// TIA Portal V20 export
VAR_GLOBAL   // PLC tag table "Unit1Em7"
   "BA030AZSBK22.00" AT %I1084.0 : Bool;   // SEPA GRIPPER CLAMP OPEN
   "BA030AZSBK22.03" AT %I1084.3 : Bool;   // SEPA GRIPPER BACKWARD
   "BA030AZSBK22.02" AT %I1084.2 : Bool;   // SEPA GRIPPER CLAMP DETECT SENSOR
   "BA030AZSBK22.10" AT %I1085.0 : Bool;   // SEPA GRIPPER CLAMP CLOSE
   "BA030AZSBK22.13" AT %I1085.3 : Bool;   // SEPA GRIPPER FORWARD
   "BA030AZSBK23.02" AT %I1088.2 : Bool;   // SEPA CUTTER UP
   "BA030AZSBK23.06" AT %I1088.6 : Bool;   // SEPA DETECT SENSOR
   "BA030AZSBK23.12" AT %I1089.2 : Bool;   // SEPA CUTTER DOWN
   "BA030AZSBK24.00" AT %I1092.0 : Bool;   // SEPA CLAMP TOP REAR UP
   "BA030AZSBK24.02" AT %I1092.2 : Bool;   // SEPA CLAMP TOP FRONT UP
   "BA030AZSBK24.04" AT %I1092.4 : Bool;   // SEPA CLAMP BTM REAR UP
   "BA030AZSBK24.06" AT %I1092.6 : Bool;   // SEPA CLAMP BTM FRONT UP
   "BA030AZSBK24.10" AT %I1093.0 : Bool;   // SEPA CLAMP TOP REAR DOWN
   "BA030AZSBK24.12" AT %I1093.2 : Bool;   // SEPA CLAMP TOP FRONT DOWN
   "BA030AZSBK24.14" AT %I1093.4 : Bool;   // SEPA CLAMP BTM REAR DOWN
   "BA030AZSBK24.16" AT %I1093.6 : Bool;   // SEPA CLAMP BTM FRONT DOWN
   "BA030AZSBK26.01" AT %I1100.1 : Bool;   // JR WINDER CLAMP TOP REAR UP/DOWN
   "BA030AZSBK26.03" AT %I1100.3 : Bool;   // JR WINDER CLAMP TOP FRONT UP/DOWN
   "BA030AZSBK26.05" AT %I1100.5 : Bool;   // JR WINDER CLAMP TOP REAR PRESSURE SWITCH
   "BA030AZSBK26.11" AT %I1101.1 : Bool;   // SPARE
   "BA030AZSBK26.13" AT %I1101.3 : Bool;   // SPARE
   "BA030AZSBK26.15" AT %I1101.5 : Bool;   // JR WINDER CLAMP TOP FRONT PRESSURE SWITCH
   "BA030AZSBK27.01" AT %I1104.1 : Bool;   // JR WINDER CLAMP BTM REAR UP/DOWN
   "BA030AZSBK27.03" AT %I1104.3 : Bool;   // JR WINDER CLAMP BTM FRONT UP/DOWN
   "BA030AZSBK27.05" AT %I1104.5 : Bool;   // JR WINDER CLAMP BTM REAR PRESSURE SWITCH
   "BA030AZSBK27.06" AT %I1104.6 : Bool;   // JR WINDER STACK DETECT SENSOR
   "BA030AZSBK27.11" AT %I1105.1 : Bool;   // SPARE
   "BA030AZSBK27.13" AT %I1105.3 : Bool;   // SPARE
   "BA030AZSBK27.15" AT %I1105.5 : Bool;   // JR WINDER CLAMP BTM FRONT PRESSURE SWITCH
   "BA030AZSBK28.02" AT %I1108.2 : Bool;   // PUSH ROLLER BACKWARD
   "BA030AZSBK28.03" AT %I1108.3 : Bool;   // PUSH ROLLER FORWARD
   "BA030AZSBK10.01" AT %I1036.1 : Bool;   // SEPA CLAMP SAFETY PIN DETECT SENSOR
   "BA030AZSBK10.11" AT %I1037.1 : Bool;   // SEPA GRIPPER SAFETY PIN DETECT SENSOR
   "BA030AZSBK10.03" AT %I1036.3 : Bool;   // SEPA CLAMP PRESSURE SWITCH
   "BA030AZSPM07.02" AT %Q2024.2 : Bool;   // JR WINDER CLAMP BTM REAR UP
   "BA030AZSPM07.03" AT %Q2024.3 : Bool;   // JR WINDER CLAMP BTM REAR DOWN
   "BA030AZSPM07.04" AT %Q2024.4 : Bool;   // JR WINDER CLAMP TOP FRONT UP
   "BA030AZSPM07.05" AT %Q2024.5 : Bool;   // JR WINDER CLAMP TOP FRONT DOWN
   "BA030AZSPM07.06" AT %Q2024.6 : Bool;   // JR WINDER CLAMP BTM FRONT UP
   "BA030AZSPM07.07" AT %Q2024.7 : Bool;   // JR WINDER CLAMP BTM FRONT DOWN
   "BA030AZSPM07.12" AT %Q2025.2 : Bool;   // PUSH ROLLER FORWARD
   "BA030AZSPM07.13" AT %Q2025.3 : Bool;   // PUSH ROLLER BACKWARD
   "BA030AZSPM03.00" AT %Q2008.0 : Bool;   // SEPA CUTTER FRONT&REAR DOWN
   "BA030AZSPM03.01" AT %Q2008.1 : Bool;   // SEPA CUTTER FRONT&REAR UP
   "BA030AZSPM03.02" AT %Q2008.2 : Bool;   // SEPA CLAMP TOP REAR DOWN
   "BA030AZSPM03.03" AT %Q2008.3 : Bool;   // SEPA CLAMP TOP REAR UP
   "BA030AZSPM03.04" AT %Q2008.4 : Bool;   // SEPA CLAMP TOP FRONT DOWN
   "BA030AZSPM03.05" AT %Q2008.5 : Bool;   // SEPA CLAMP TOP FRONT UP
   "BA030AZSPM03.06" AT %Q2008.6 : Bool;   // SEPA CLAMP BTM REAR DOWN
   "BA030AZSPM03.07" AT %Q2008.7 : Bool;   // SEPA CLAMP BTM REAR UP
   "BA030AZSPM03.10" AT %Q2009.0 : Bool;   // SEPA CLAMP BTM FRONT DOWN
   "BA030AZSPM03.11" AT %Q2009.1 : Bool;   // SEPA CLAMP BTM FRONT UP
   "BA030AZSPM03.12" AT %Q2009.2 : Bool;   // SEPA GRIPPER CLOSE
   "BA030AZSPM03.13" AT %Q2009.3 : Bool;   // SEPA GRIPPER OPEN
   "BA030AZSPM03.14" AT %Q2009.4 : Bool;   // SEPA GRIPPER FORWARD
   "BA030AZSPM03.15" AT %Q2009.5 : Bool;   // SEPA GRIPPER BACKWARD
   "BA030AZSPM07.00" AT %Q2024.0 : Bool;   // JR WINDER CLAMP TOP REAR UP
   "BA030AZSPM07.01" AT %Q2024.1 : Bool;   // JR WINDER CLAMP TOP REAR DOWN
END_VAR
VAR_GLOBAL CONSTANT   // user constants
   U1EM7_JOB01 : DInt := 1;
   U1EM7_JOB02 : DInt := 2;
   U1EM7_JOB03 : DInt := 3;
   U1EM7_JOB04 : DInt := 4;
   U1EM7_JOB05 : DInt := 5;
   U1EM7_JOB06 : DInt := 6;
   U1EM7_JOB07 : DInt := 7;
   U1EM7_JOB08 : DInt := 8;
   U1EM7_JOB09 : DInt := 9;
   U1EM7_JOB10 : DInt := 10;
   U1EM7_JOB11 : DInt := 11;
   U1EM7_JOB12 : DInt := 12;
   U1EM7_JOB13 : DInt := 13;
   U1EM7_JOB14 : DInt := 14;
   U1EM7_JOB15 : DInt := 15;
   U1EM7_JOB16 : DInt := 16;
   U1EM7_JOB17 : DInt := 17;
   U1EM7_JOB18 : DInt := 18;
   U1EM7_JOB19 : DInt := 19;
   U1EM7_JOB20 : DInt := 20;
   U1EM7_JOB21 : DInt := 21;
   U1EM7_JOB22 : DInt := 22;
   U1EM7_JOB23 : DInt := 23;
   U1EM7_JOB24 : DInt := 24;
   U1EM7_JOB25 : DInt := 25;
   U1EM7_JOB26 : DInt := 26;
   U1EM7_JOB27 : DInt := 27;
   U1EM7_JOB28 : DInt := 28;
   U1EM7_JOB29 : DInt := 29;
   U1EM7_JOB30 : DInt := 30;
   U1EM7_JOB31 : DInt := 31;
   U1EM7_JOB32 : DInt := 32;
   U1EM7_JOB33 : DInt := 33;
   U1EM7_JOB34 : DInt := 34;
   U1EM7_JOB35 : DInt := 35;
   U1EM7_JOB36 : DInt := 36;
   U1EM7_JOB37 : DInt := 37;
   U1EM7_JOB38 : DInt := 38;
   U1EM7_JOB39 : DInt := 39;
   U1EM7_JOB40 : DInt := 40;
   U1EM7_JOB41 : DInt := 41;
   U1EM7_JOB42 : DInt := 42;
   U1EM7_JOB43 : DInt := 43;
   U1EM7_JOB44 : DInt := 44;
   U1EM7_JOB45 : DInt := 45;
   U1EM7_JOB46 : DInt := 46;
   U1EM7_JOB47 : DInt := 47;
   U1EM7_JOB48 : DInt := 48;
   U1EM7_JOB49 : DInt := 49;
   U1EM7_JOB50 : DInt := 50;
   U1EM7_JOB51 : DInt := 51;
   U1EM7_JOB52 : DInt := 52;
   U1EM7_JOB53 : DInt := 53;
   U1EM7_JOB54 : DInt := 54;
   U1EM7_JOB55 : DInt := 55;
   U1EM7_JOB56 : DInt := 56;
   U1EM7_JOB57 : DInt := 57;
   U1EM7_JOB58 : DInt := 58;
   U1EM7_JOB59 : DInt := 59;
   U1EM7_JOB60 : DInt := 60;
   U1EM7_JOB61 : DInt := 61;
   U1EM7_JOB62 : DInt := 62;
   U1EM7_JOB63 : DInt := 63;
   U1EM7_JOB64 : DInt := 64;
   U1EM7_JOB65 : DInt := 65;
   U1EM7_JOB66 : DInt := 66;
   U1EM7_JOB67 : DInt := 67;
   U1EM7_JOB68 : DInt := 68;
   U1EM7_JOB69 : DInt := 69;
   U1EM7_JOB70 : DInt := 70;
   U1EM7_JOB71 : DInt := 71;
   U1EM7_JOB72 : DInt := 72;
   U1EM7_JOB73 : DInt := 73;
   U1EM7_JOB74 : DInt := 74;
   U1EM7_JOB75 : DInt := 75;
   U1EM7_JOB76 : DInt := 76;
   U1EM7_JOB77 : DInt := 77;
   U1EM7_JOB78 : DInt := 78;
   U1EM7_JOB79 : DInt := 79;
   U1EM7_JOB80 : DInt := 80;
   U1EM7_JOB81 : DInt := 81;
   U1EM7_JOB82 : DInt := 82;
   U1EM7_JOB83 : DInt := 83;
   U1EM7_JOB84 : DInt := 84;
   U1EM7_JOB85 : DInt := 85;
   U1EM7_JOB86 : DInt := 86;
   U1EM7_JOB87 : DInt := 87;
   U1EM7_JOB88 : DInt := 88;
   U1EM7_JOB89 : DInt := 89;
   U1EM7_JOB90 : DInt := 90;
   U1EM7_JOB91 : DInt := 91;
   U1EM7_JOB92 : DInt := 92;
   U1EM7_JOB93 : DInt := 93;
   U1EM7_JOB94 : DInt := 94;
   U1EM7_JOB95 : DInt := 95;
   U1EM7_JOB96 : DInt := 96;
   U1EM7_JOB97 : DInt := 97;
   U1EM7_JOB98 : DInt := 98;
   U1EM7_JOB99 : DInt := 99;
   U1EM7_SEQUENCE01 : Int := 1;
   U1EM7_SEQUENCE02 : Int := 2;
   U1EM7_SEQUENCE03 : Int := 3;
   U1EM7_SEQUENCE04 : Int := 4;
   U1EM7_SEQUENCE05 : Int := 5;
   U1EM7_SEQUENCE06 : Int := 6;
   U1EM7_SEQUENCE07 : Int := 7;
   U1EM7_SEQUENCE08 : Int := 8;
   U1EM7_SEQUENCE09 : Int := 9;
   U1EM7_SEQUENCE10 : Int := 10;
   U1EM7_SEQUENCE11 : Int := 11;
   U1EM7_SEQUENCE12 : Int := 12;
   U1EM7_SEQUENCE13 : Int := 13;
   U1EM7_SEQUENCE14 : Int := 14;
   U1EM7_SEQUENCE15 : Int := 15;
   U1EM7_SEQUENCE16 : Int := 16;
   U1EM7_SEQUENCE17 : Int := 17;
   U1EM7_SEQUENCE18 : Int := 18;
   U1EM7_SEQUENCE19 : Int := 19;
   U1EM7_SEQUENCE20 : Int := 20;
   U1EM7_SEQUENCE21 : Int := 21;
   U1EM7_SEQUENCE22 : Int := 22;
   U1EM7_SEQUENCE23 : Int := 23;
   U1EM7_SEQUENCE24 : Int := 24;
   U1EM7_SEQUENCE25 : Int := 25;
   U1EM7_SEQUENCE26 : Int := 26;
   U1EM7_SEQUENCE27 : Int := 27;
   U1EM7_SEQUENCE28 : Int := 28;
   U1EM7_SEQUENCE29 : Int := 29;
   U1EM7_SEQUENCE30 : Int := 30;
   U1EM7_SEQUENCE31 : Int := 31;
   U1EM7_SEQUENCE32 : Int := 32;
   U1EM7_SEQUENCE33 : Int := 33;
   U1EM7_SEQUENCE34 : Int := 34;
   U1EM7_SEQUENCE35 : Int := 35;
   U1EM7_SEQUENCE36 : Int := 36;
   U1EM7_SEQUENCE37 : Int := 37;
   U1EM7_SEQUENCE38 : Int := 38;
   U1EM7_SEQUENCE39 : Int := 39;
   U1EM7_SEQUENCE40 : Int := 40;
   U1EM7_SEQUENCE41 : Int := 41;
   U1EM7_SEQUENCE42 : Int := 42;
   U1EM7_SEQUENCE43 : Int := 43;
   U1EM7_SEQUENCE44 : Int := 44;
   U1EM7_SEQUENCE45 : Int := 45;
   U1EM7_SEQUENCE46 : Int := 46;
   U1EM7_SEQUENCE47 : Int := 47;
   U1EM7_SEQUENCE48 : Int := 48;
   U1EM7_SEQUENCE49 : Int := 49;
   U1EM7_SEQUENCE50 : Int := 50;
   U1EM7_SEQUENCE51 : Int := 51;
   U1EM7_SEQUENCE52 : Int := 52;
   U1EM7_SEQUENCE53 : Int := 53;
   U1EM7_SEQUENCE54 : Int := 54;
   U1EM7_SEQUENCE55 : Int := 55;
   U1EM7_SEQUENCE56 : Int := 56;
   U1EM7_SEQUENCE57 : Int := 57;
   U1EM7_SEQUENCE58 : Int := 58;
   U1EM7_SEQUENCE59 : Int := 59;
   U1EM7_SEQUENCE60 : Int := 60;
   U1EM7_SEQUENCE61 : Int := 61;
   U1EM7_SEQUENCE62 : Int := 62;
   U1EM7_SEQUENCE63 : Int := 63;
   U1EM7_SEQUENCE64 : Int := 64;
   U1EM7_SEQUENCE65 : Int := 65;
   U1EM7_SEQUENCE66 : Int := 66;
   U1EM7_SEQUENCE67 : Int := 67;
   U1EM7_SEQUENCE68 : Int := 68;
   U1EM7_SEQUENCE69 : Int := 69;
   U1EM7_SEQUENCE70 : Int := 70;
   U1EM7_SEQUENCE71 : Int := 71;
   U1EM7_SEQUENCE72 : Int := 72;
   U1EM7_SEQUENCE73 : Int := 73;
   U1EM7_SEQUENCE74 : Int := 74;
   U1EM7_SEQUENCE75 : Int := 75;
   U1EM7_SEQUENCE76 : Int := 76;
   U1EM7_SEQUENCE77 : Int := 77;
   U1EM7_SEQUENCE78 : Int := 78;
   U1EM7_SEQUENCE79 : Int := 79;
   U1EM7_SEQUENCE80 : Int := 80;
   U1EM7_SEQUENCE81 : Int := 81;
   U1EM7_SEQUENCE82 : Int := 82;
   U1EM7_SEQUENCE83 : Int := 83;
   U1EM7_SEQUENCE84 : Int := 84;
   U1EM7_SEQUENCE85 : Int := 85;
   U1EM7_SEQUENCE86 : Int := 86;
   U1EM7_SEQUENCE87 : Int := 87;
   U1EM7_SEQUENCE88 : Int := 88;
   U1EM7_SEQUENCE89 : Int := 89;
   U1EM7_SEQUENCE90 : Int := 90;
   U1EM7_SEQUENCE91 : Int := 91;
   U1EM7_SEQUENCE92 : Int := 92;
   U1EM7_SEQUENCE93 : Int := 93;
   U1EM7_SEQUENCE94 : Int := 94;
   U1EM7_SEQUENCE95 : Int := 95;
   U1EM7_SEQUENCE96 : Int := 96;
   U1EM7_SEQUENCE97 : Int := 97;
   U1EM7_SEQUENCE98 : Int := 98;
   U1EM7_SEQUENCE99 : Int := 99;
   U1EM7_NO_OF_SEQUENCE : USInt := 3;
   U1EM7_NO_OF_AXES : USInt := 9;
   U1EM7_NO_OF_CAM : USInt := 6;
END_VAR
